// TIA Portal V17 export
// export: Created 2023-10-17T06:55:21.2801052Z, ExportSetting WithDefaults, DisplayName Totally Integrated Automation Portal, DisplayVersion V17, DisplayName TIA Portal Openness, DisplayVersion V17, DisplayName TIA Portal Version Control Interface, DisplayVersion V17, DisplayName STEP 7 Professional, DisplayVersion V17, DisplayName STEP 7 Safety, DisplayVersion V17, DisplayName WinCC Advanced, DisplayVersion V17
VAR_GLOBAL   // PLC tag table "Default tag table"
   Batch_WeightScale_Done AT %M2.2 : Bool;
   Batch_FillToMixer_Done AT %M2.3 : Bool;
   Batch_Mixing_Done AT %M2.4 : Bool;
   Batch_Fillto_Pasteurisation_Done AT %M2.5 : Bool;
   Batch_Pasteurizing_Done AT %M2.6 : Bool;
   Filler_Ready AT %M2.7 : Bool;
   Clock_Byte AT %MB0 : Byte;
   Clock_10Hz AT %M0.0 : Bool;
   Clock_5Hz AT %M0.1 : Bool;
   "Clock_2.5Hz" AT %M0.2 : Bool;
   Clock_2Hz AT %M0.3 : Bool;
   "Clock_1.25Hz" AT %M0.4 : Bool;
   Clock_1Hz AT %M0.5 : Bool;
   "Clock_0.625Hz" AT %M0.6 : Bool;
   "Clock_0.5Hz" AT %M0.7 : Bool;
END_VAR
